FUNCTION_BLOCK Hopper_Level
VAR_INPUT
	HopperLevel_Input:WORD;
END_VAR
VAR_OUTPUT
	HopperLevel_PCT:REAL;
END_VAR
VAR
	HopperLevel_Real: REAL;
END_VAR

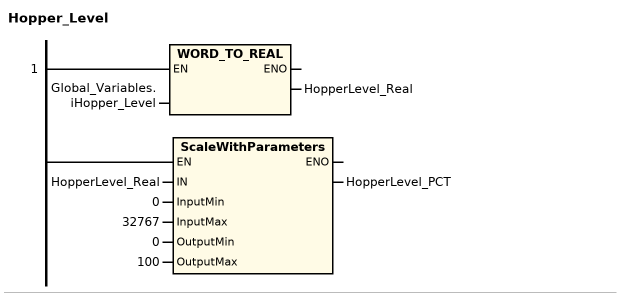
// NETWORK 1
HopperLevel_Real := WORD_TO_REAL(Global_Variables.iHopper_Level);
HopperLevel_PCT := ScaleWithParameters(IN := HopperLevel_Real, InputMin := 0, InputMax := 32767, OutputMin := 0, OutputMax := 100);

END_FUNCTION_BLOCK

(* stored: Version 1.1.0.1, ProductVersion 3.1.4024.15
   POU Hopper_Level: Id {4e081826-ef39-4b89-8bc3-f919449fa25e}, SpecialFunc None *)
